// TwinCAT 3 PLC project PackML_V2
// ProgramVersion: 3.1.4022.4
// libraries:
//   Tc2_MC2, * (Beckhoff Automation GmbH)
//   Tc2_Standard, * (Beckhoff Automation GmbH)
//   Tc2_System, * (Beckhoff Automation GmbH)
//   Tc3_Module, * (Beckhoff Automation GmbH)
//   Tc3_mxAutomation, * (Beckhoff Automation GmbH)
//   Tc3_PackML_V2, * (Beckhoff Automation GmbH)
// project tree:
//   DUTs/ Button.TcDUT
//   GVLs/ CONST_GV.TcGVL, GV.TcGVL, PERS_GV.TcGVL, SIGNAL.TcDUT
//   / PlcTask.TcTTO
//   POUs/ MAIN.TcPOU
//   POUs/Unit/ PackagingMachine.TcPOU, Robot.TcPOU, UnitBaseClass.TcPOU
// real-time tasks:
//   TASK PlcTask: cycle T#10ms, priority 20, ADS port 350

CONFIGURATION PackML_V2
    RESOURCE PLC ON TwinCAT3
        TASK PlcTask(INTERVAL := T#10ms, PRIORITY := 20);
        PROGRAM MAIN WITH PlcTask : MAIN;
    END_RESOURCE
END_CONFIGURATION

// ---- DUTs/Button.TcDUT
// struct for command buttons (kapula)
TYPE Button :
STRUCT
	isPressed	AT	%I*	:	BIT;
	isLit		AT	%Q*	:	BOOL;
END_STRUCT
END_TYPE

// ---- GVLs/SIGNAL.TcDUT

// enum for user triggered signals (buttons)
TYPE SIGNAL:
(
	noSignal 		:= 	-1,
	
	// command signals (triggered from kapula)
	resetSignal		:=	0,
	startSignal		:= 	1,
	stopSignal		:= 	2,
	holdSignal		:= 	3,
	unHoldSignal	:=	4,
	suspendSignal	:=	5,
	unSuspendSignal	:=	6,
	abortSignal		:=	7,	
	clearSignal		:= 	8,
	
	// unit mode signals (to be decided how to trigger)
	productionModeSignal	:= 	9,
	maintenanceModeSignal	:=	10,
	manualModeSignal		:=	11
);
END_TYPE

// ---- GVLs/CONST_GV.TcGVL
{attribute 'qualified_only'}
VAR_GLOBAL CONSTANT
	nSubUnits	:	UINT		:=	1;
	
END_VAR

// ---- GVLs/GV.TcGVL
VAR_GLOBAL
	packTags	:	ST_PackMLv30;
END_VAR

// ---- GVLs/PERS_GV.TcGVL
{attribute 'qualified_only'}
VAR_GLOBAL PERSISTENT
	// only first three axises available
	 //R1	:	AXIS_REF;
	 //R2	:	AXIS_REF;
	 //R3	:	AXIS_REF;
	// R4	:	AXIS_REF;
	// R5	:	AXIS_REF;
	// R6	:	AXIS_REF;
END_VAR

// ---- POUs/MAIN.TcPOU
PROGRAM MAIN
VAR
	
	running				:	BOOL	:= FALSE;
	packagingMachine	:	PackagingMachine;
	input				:	BOOL;
	
END_VAR

// ready when packagingmachine is initialized
// initialized when in stopped state and modemanager enabled
IF NOT running THEN
	IF machineConfig() THEN
		running := TRUE;
	ELSE
		// configurationError
	END_IF
	
ELSE
	CASE packagingMachine.getSignal() OF
		noSignal:
			packagingMachine();
			
		startSignal:
			packagingMachine.setState(command:=ePMLCommand_Start);
			
		stopSignal:
			packagingMachine.setState(command:=ePMLCommand_Stop);
		
		abortSignal:
			packagingMachine.setState(command:=ePMLCommand_Abort);
				
		resetSignal:
			packagingMachine.setState(command:=ePMLCommand_Reset);
			
		clearSignal:
			packagingMachine.setState(command:=ePMLCommand_Clear);

		productionModeSignal:
			packagingMachine.setMode(modeCommand:=ePMLProtUnitMode_Production);
			
		maintenanceModeSignal:
			packagingMachine.setMode(modeCommand:=ePMLProtUnitMode_Maintenance);
			
		manualModeSignal:
			packagingMachine.setMode(modeCommand:=ePMLProtUnitMode_Manual);
			
	END_CASE
	
END_IF

// machine config is used to initialize all units.

METHOD machineConfig : BOOL
VAR_INPUT
END_VAR
VAR
	initMode		:	E_PMLProtectedUnitMode	:= 	ePMLProtUnitMode_Production;
	initCommand		:	E_PMLCommand			:=	ePMLCommand_Stop;
	
	subUnits	:	ARRAY[1..CONST_GV.nSubUnits] OF UnitBaseClass;
	staubli		:	Robot;
END_VAR

// 		subUnit1 - Staubli
subUnits[1] := staubli;


// 		subUnit2 ... subUnitn
// subUnits[2] := subUnit2;


// initialize
packagingMachine.initialize(arg1	:=	initMode, 
							arg2	:=	initCommand, 
							arg3	:=	ADR(subUnits));

							
// return initialization status							
machineConfig := packagingMachine.initialized;
END_METHOD

END_PROGRAM

// ---- POUs/Unit/PackagingMachine.TcPOU
// PackagingMachine object represents the packaging machine as a whole.

// right now though the packaging machine only consists of staubli robot,
// but in future projects of extending the system it is now "easy" to do so.

FUNCTION_BLOCK PackagingMachine EXTENDS UnitBaseClass
VAR_INPUT
	// reset button
	resetButton		:	Button;
	// start button
	startButton		:	Button;	
	// stop button
	stopButton		:	Button;
	// emergency stop
	abortButton		:	BOOL;
	// clear emergency stop 
	clearButton		:	BOOL;
	
	(* not connected to IO
	holdButton		:	Button;
	unHoldButton	:	Button;
	suspendButton	:	Button;
	unSuspendButton	:	Button
	*)

	// mode change buttons (do not exist in real life)
	productionModeButton	:	BIT;
	maintenanceModeButton	:	BIT;
	manualModeButton		:	BIT;	
END_VAR
VAR_OUTPUT
END_VAR
VAR
	subUnits	:	POINTER TO ARRAY[1..CONST_GV.nSubUnits] OF UnitBaseClass;
END_VAR

METHOD getSignal : INT
VAR_INPUT
END_VAR

// arranged in a way that most important ones are checked first.

// probably needs more conditions than just button signal pressed. 
// for example the statements should be ignored if machine in transition state etc.

IF abortButton THEN
	getSignal := abortSignal;
	RETURN;
END_IF

//in currently in active state (starting, stopping, etc..) ignore
IF inStateTransition THEN
	RETURN;
END_IF
	
IF stopButton.isPressed THEN
	getSignal := stopSignal;
	RETURN;
	
ELSIF startButton.isPressed THEN
	getSignal := startSignal;
	RETURN;
	
ELSIF resetButton.isPressed THEN
	getSignal := resetSignal;
	RETURN;
	
ELSIF clearButton THEN
	getSignal := clearSignal;
	RETURN;

(*	
ELSIF holdButton.isPressed THEN
	getSignal := holdSignal;
	RETURN;
	
ELSIF unHoldButton.isPressed THEN
	getSignal := unHoldSignal;
	RETURN;
	
ELSIF suspendButton.isPressed THEN
	getSignal := suspendSignal;
	RETURN;
	
ELSIF unSuspendButton.isPressed THEN
	getSignal := unSuspendSignal;
	RETURN;
*)

ELSIF productionModeButton THEN
	getSignal := productionModeSignal;
	RETURN;
	
ELSIF maintenanceModeButton THEN
	getSignal := maintenanceModeSignal;
	RETURN;
	
ELSIF manualModeButton THEN
	getSignal := manualModeSignal;
	RETURN;
	
ELSE
	getSignal := -1;
	
END_IF
END_METHOD

METHOD initialize	:	BOOL
VAR_INPUT
	arg1 	:	E_PMLProtectedUnitMode;
	arg2	:	E_PMLCommand;
	arg3	:	POINTER TO ARRAY[1..CONST_GV.nSubUnits] OF UnitBaseClass;
END_VAR
VAR
	i	:	UINT;
END_VAR
// initialize sub units
FOR i:=1 TO CONST_GV.nSubUnits BY 1 DO
	// if any of the sub units is uninitialized then the whole machine is too
	IF NOT arg3^[i].initialize(arg1:=arg1, arg2:=arg2, arg3:=0) THEN
		RETURN;
	END_IF
END_FOR

// initialize self
unitModeManager.bExecute := TRUE;
IF (NOT (SUPER^.setMode(modeCommand:=arg1) AND SUPER^.setState(command := arg2)) ) THEN
	unitModeManager.bExecute := FALSE;
	RETURN;
END_IF

resetButton.isLit 				:= TRUE;
startButton.isLit 				:= TRUE;
stopButton.isLit				:= TRUE;

THIS^.subUnits 					:= arg3;
THIS^.initialized 				:= TRUE;
initialize 						:= TRUE;
END_METHOD

METHOD setMode : BOOL
VAR_INPUT
	modeCommand	:	DINT;
END_VAR
VAR
	prevMode	:	E_PMLProtectedUnitMode;
	i			:	UINT;
END_VAR
// if any of the subUnits cannot change mode to given mode return false
FOR i:=1 TO CONST_GV.nSubUnits BY 1 DO
	IF NOT subUnits^[i].setMode(modeCommand:=modeCommand) THEN
		setMode := FALSE;
		RETURN;
	END_IF
END_FOR
SUPER^.setMode(modeCommand:=modeCommand);
setMode := TRUE;
END_METHOD


// setState method. Attempts to change the state of unit according to 
// the given input command which is a result of received user signal (startButton, stopButton ... ).

(* possible commands :	
	ePMLCommand_Undefined   := 0,
	ePMLCommand_Reset       := 1,
	ePMLCommand_Start       := 2,
	ePMLCommand_Stop        := 3,
	ePMLCommand_Hold        := 4,
	ePMLCommand_Unhold      := 5,
	ePMLCommand_Suspend     := 6,
	ePMLCommand_Unsuspend   := 7,
	ePMLCommand_Abort       := 8,
	ePMLCommand_Clear       := 9
*)

METHOD setState : BOOL
VAR_INPUT
	command	:	E_PMLCommand;
END_VAR
VAR
	prevState	:	E_PMLState;
	i			:	UINT;
END_VAR
// if any of the subUnits cannot change state to given state return false
FOR i:=1 TO CONST_GV.nSubUnits BY 1 DO
	IF NOT subUnits^[i].setState(command:=command) THEN
		setState := FALSE;
		RETURN;
	END_IF
END_FOR
SUPER^.setState(command:=command);
setState := TRUE;
END_METHOD

END_FUNCTION_BLOCK

// ---- POUs/Unit/UnitBaseClass.TcPOU

// BASE CLASS FOR EVERY UNIT/MACHINE IN THE SYSTEM
	// consists of modemanager, statemachine, UnitState interface
	// and setMode and setState methods.
	
	
FUNCTION_BLOCK UnitBaseClass IMPLEMENTS ITF_UnitState
VAR_INPUT

END_VAR
VAR_OUTPUT
	currentMode		:	DINT;
	currentState	:	E_PMLState;
	initialized		:	BOOL;
END_VAR
VAR
	unitModeManager		:	PML_UnitModeManager;
	stateMachine		:	PML_StateMachine;
	inModeTransition	:	BOOL	:=	FALSE;
	inStateTransition	:	BOOL	:= 	FALSE;
END_VAR

// method for checking if command is already being executed/has been executed
// for example if currentState is stopped then stop command is called
// this method returns true and nothing happens in setState method (where this method is called)

METHOD alreadyActive : BOOL
VAR_INPUT
	command 		:	E_PMLCommand;
	currentState	:	E_PMLState;
END_VAR

(* possible commands :	
	ePMLCommand_Undefined   := 0,
	ePMLCommand_Reset       := 1,
	ePMLCommand_Start       := 2,
	ePMLCommand_Stop        := 3,
	ePMLCommand_Hold        := 4,
	ePMLCommand_Unhold      := 5,
	ePMLCommand_Suspend     := 6,
	ePMLCommand_Unsuspend   := 7,
	ePMLCommand_Abort       := 8,
	ePMLCommand_Clear       := 9
*)

CASE command OF
	0: 	IF currentState = ePMLState_Undefined THEN
			alreadyActive := TRUE;
		END_IF		
	
	1: 	IF currentState = ePMLState_Resetting OR currentState = ePMLState_Idle THEN
			alreadyActive := TRUE;
		END_IF
		
	2: IF currentState = ePMLState_Starting OR currentState = ePMLState_Execute THEN
			alreadyActive := TRUE;
		END_IF
	
	3: 	IF currentState = ePMLState_Stopping OR currentState = ePMLState_Stopped THEN
			alreadyActive := TRUE;
		END_IF
	
	4: 	IF currentState = ePMLState_Holding OR currentState = ePMLState_Held THEN
			alreadyActive := TRUE;
		END_IF
	
	5: 	IF currentState = ePMLState_UnHolding OR currentState = ePMLState_Execute THEN
			alreadyActive := TRUE;
		END_IF
	
	6: 	IF currentState = ePMLState_Suspending OR currentState = ePMLState_Suspended THEN
			alreadyActive := TRUE;
		END_IF
	
	7: 	IF currentState = ePMLState_Unsuspending OR currentState = ePMLState_Execute THEN
			alreadyActive := TRUE;
		END_IF
	
	8: 	IF currentState = ePMLState_Aborting OR currentState = ePMLState_Aborted THEN
			alreadyActive := TRUE;
		END_IF
	
	9:	IF currentState = ePMLState_Clearing OR currentState = ePMLState_Stopped THEN
			alreadyActive := TRUE;
		END_IF 	
END_CASE
END_METHOD

METHOD initialize	:	BOOL
VAR_INPUT
	arg1 	:	E_PMLProtectedUnitMode; 	// 	unitModeCommand
	arg2	:	E_PMLCommand;				//	command
	arg3	:	POINTER TO ARRAY[1..CONST_GV.nSubUnits] OF UnitBaseClass := 0; // subUnits
END_VAR
unitModeManager.bExecute := TRUE;

IF (NOT (THIS^.setMode(modeCommand:=arg1) AND THIS^.setState(command := arg2)) ) THEN
	// set initialized
	unitModeManager.bExecute := FALSE;
	RETURN;
END_IF

// instance property
THIS^.initialized := TRUE;
// method return value
initialize := TRUE;
END_METHOD


METHOD M_Aborted
END_METHOD

// M_Aborting is an 'acting' type state called in UnitBaseClass::setState()
// due to rising signal of emergency stop button.

// the implementation is done in derived classes
METHOD M_Aborting
M_StateComplete();
END_METHOD

{warning 'add method implementation'}
METHOD M_Clearing
M_StateComplete();
END_METHOD

{warning 'add method implementation'}
METHOD M_Complete
END_METHOD

{warning 'add method implementation'}
METHOD M_Completing
M_StateComplete();
END_METHOD

{warning 'add method implementation'}
METHOD M_Execute
END_METHOD

{warning 'add method implementation'}
METHOD M_Held
END_METHOD

{warning 'add method implementation'}
METHOD M_Holding
M_StateComplete();
END_METHOD

{warning 'add method implementation'}
METHOD M_Idle
END_METHOD

{warning 'add method implementation'}
METHOD M_Resetting
M_StateComplete();
END_METHOD

{warning 'add method implementation'}
METHOD M_Starting
M_StateComplete();
END_METHOD


// PML_StateMachine::M_StateCompleted() is what actually 
// changes the state from acting state to wait state.
// that's why this method is called after every '-ing' (acting) state.

METHOD M_StateComplete
stateMachine.M_StateComplete();
currentState := stateMachine.eState;
inStateTransition := FALSE;
END_METHOD

{warning 'add method implementation'}
METHOD M_Stopped
END_METHOD

{warning 'add method implementation'}
METHOD M_Stopping
M_StateComplete();
END_METHOD

{warning 'add method implementation'}
METHOD M_Suspended
END_METHOD

{warning 'add method implementation'}
METHOD M_Suspending
M_StateComplete();
END_METHOD

{warning 'add method implementation'}
METHOD M_Undefined
END_METHOD

{warning 'add method implementation'}
METHOD M_Unholding
M_StateComplete();
END_METHOD

{warning 'add method implementation'}
METHOD M_Unsuspending
M_StateComplete();
END_METHOD

METHOD setMode : BOOL
VAR_INPUT
	modeCommand	:	DINT;
END_VAR
VAR
	prevMode	:	E_PMLProtectedUnitMode;
END_VAR
// check if tryign to cahnge mode to one that is already active
IF modeCommand = currentMode THEN
	setMode := TRUE;
	RETURN;
END_IF

// save current mode as previous mode
prevMode := currentMode;

// update current mode
unitModeManager(eModeCommand := modeCommand, 
				eState := currentState,
				eModeStatus => currentMode);
				
// check if mode was changed, if not return false
IF(currentMode = prevMode) OR (currentMode = ePMLProtUnitMode_Invalid) THEN
	setMode := FALSE;
	RETURN;
END_IF

setMode := TRUE;
END_METHOD


// setState method. Attempts to change the state of unit according to 
// the given input command which is a result of received user signal (startButton, stopButton ... ).


METHOD setState : BOOL
VAR_INPUT
	command	:	E_PMLCommand;
END_VAR
VAR
	prevState	:	E_PMLState;	
END_VAR

(* possible commands :	
	ePMLCommand_Undefined   := 0,
	ePMLCommand_Reset       := 1,
	ePMLCommand_Start       := 2,
	ePMLCommand_Stop        := 3,
	ePMLCommand_Hold        := 4,
	ePMLCommand_Unhold      := 5,
	ePMLCommand_Suspend     := 6,
	ePMLCommand_Unsuspend   := 7,
	ePMLCommand_Abort       := 8,
	ePMLCommand_Clear       := 9
*)
// for example if currentState is starting and start button 
// is pressed nothing happens
IF alreadyActive(command:=command, currentState:=currentState) THEN
	setState := TRUE;
	RETURN;
END_IF

// save current state as previous state
prevState := currentState;

// update current state
stateMachine(eMode:=currentMode, eCommand:=command, eState=>currentState);

// check whether the state was changed, if not return false
IF (currentState = prevState) OR (currentState = ePMLState_Undefined) THEN
	setState := FALSE;
	RETURN;
END_IF

inStateTransition := TRUE;
setState := TRUE;

// run resulted state method.
CASE currentState OF	
	ePMLState_Undefined:
		M_Undefined();
	
	ePMLState_Resetting:
		M_Resetting();
		
    ePMLState_Starting:
		M_Starting();		
		
    ePMLState_Stopping:
		M_Stopping();
		
    ePMLState_Aborting:
		M_Aborting();
		
    ePMLState_Holding:
		M_Holding();
		
    ePMLState_Unholding:
		M_Unholding();
		
    ePMLState_Suspending:
		M_Suspending();
		
    ePMLState_Unsuspending:
		M_Unsuspending();		
		
	ePMLState_Clearing:
		M_Clearing();		
END_CASE
END_METHOD

END_FUNCTION_BLOCK

// ---- POUs/Unit/Robot.TcPOU

// class for robot units.
FUNCTION_BLOCK Robot EXTENDS UnitBaseClass
VAR_INPUT
	//axes		:	ST_KinAxes;
END_VAR
VAR_OUTPUT
	pos		:	E6POS;
END_VAR
VAR
	//power	:	MC_Power;
	//status	:	ST_AxisStatus;
END_VAR

METHOD fkine : BOOL
VAR_INPUT
END_VAR
END_METHOD

METHOD ikine : BOOL
VAR_INPUT
END_VAR
END_METHOD

METHOD initialize	:	BOOL
VAR_INPUT
	arg1 	:	E_PMLProtectedUnitMode;
	arg2	:	E_PMLCommand;
	arg3	:	POINTER TO ARRAY[1..CONST_GV.nSubUnits] OF UnitBaseClass;
END_VAR
SUPER^.initialize(arg1:=arg1, arg2:=arg2, arg3:=0);

// initialize axis etc
END_METHOD

METHOD moveFree : BOOL
VAR_INPUT
END_VAR
END_METHOD

METHOD moveLinear : BOOL
VAR_INPUT
END_VAR
END_METHOD

END_FUNCTION_BLOCK
